FUNCTION TryConvert_LREAL_TO_UDINT : BOOL
VAR_INPUT
	in : LREAL;
	out : REFERENCE TO UDINT;
END_VAR

IF in > DatatypeLimits.MAX_VALUE_OF_LREAL_WHICH_CAN_BE_HELD_IN_A_UDINT THEN
	RETURN;
END_IF

IF in < DatatypeLimits.MIN_VALUE_OF_LREAL_WHICH_CAN_BE_HELD_IN_A_UDINT THEN
	RETURN;
END_IF

out := LREAL_TO_UDINT(in);
TryConvert_LREAL_TO_UDINT := TRUE;

END_FUNCTION

(* stored: Version 1.1.0.1, ProductVersion 3.1.4024.12
   POU TryConvert_LREAL_TO_UDINT: Id {68429051-77fd-4ba7-9aa3-fbf8511d58ce}, SpecialFunc None *)
